(* IEC 61131-3 sources: MotorControl/, 1 file *)

(* ---- MotorControl.st ---- *)
PROGRAM MotorControl
VAR
    motorStart : BOOL := FALSE; (* Motor start command *)
    motorStop : BOOL := FALSE;  (* Motor stop command *)
    motorRunning : BOOL := FALSE; (* Motor running status *)
END_VAR

(* Motor control logic *)
IF motorStart THEN
    motorRunning := TRUE;
ELSIF motorStop THEN
    motorRunning := FALSE;
END_IF

(* Monitoring motor status *)
IF motorRunning THEN
    (* Add code to monitor motor parameters, e.g., speed, temperature *)
END_IF
